(* CoDeSys 2.3 export: SCHU-P2-3.EXP *)

(* POU MAIN, CFC *)
PROGRAM MAIN
VAR
	TCT: ISTOK_TaskCycleTime;
END_VAR
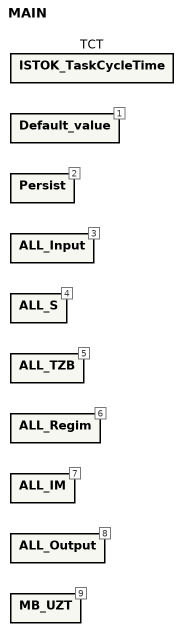
_CFC_ (* Continuous Function Chart, elements in execution order *)
#0 TCT:ISTOK_TaskCycleTime()
#1 Default_value()
#2 Persist()
#3 ALL_Input()
#4 ALL_S()
#5 ALL_TZB()
#6 ALL_Regim()
#7 ALL_IM()
#8 ALL_Output()
#9 MB_UZT()
_END_CFC_
(* the same logic as Structured Text *)
TCT();
Default_value();
Persist();
ALL_Input();
ALL_S();
ALL_TZB();
ALL_Regim();
ALL_IM();
ALL_Output();
MB_UZT();
END_PROGRAM

(* POU Lib/ISTOK_TaskCycleTime, CFC *)
FUNCTION_BLOCK ISTOK_TaskCycleTime
VAR_INPUT
END_VAR
VAR_OUTPUT
END_VAR
VAR
END_VAR
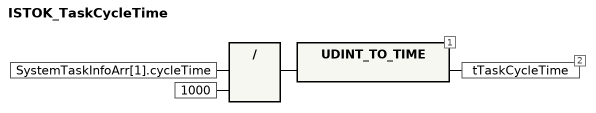
_CFC_ (* Continuous Function Chart, elements in execution order *)
#0 /(SystemTaskInfoArr[1].cycleTime, 1000)
#1 UDINT_TO_TIME(#0)
#2 tTaskCycleTime <= #1
_END_CFC_
END_FUNCTION_BLOCK

(* POU Default_value, CFC *)
PROGRAM Default_value
VAR
END_VAR
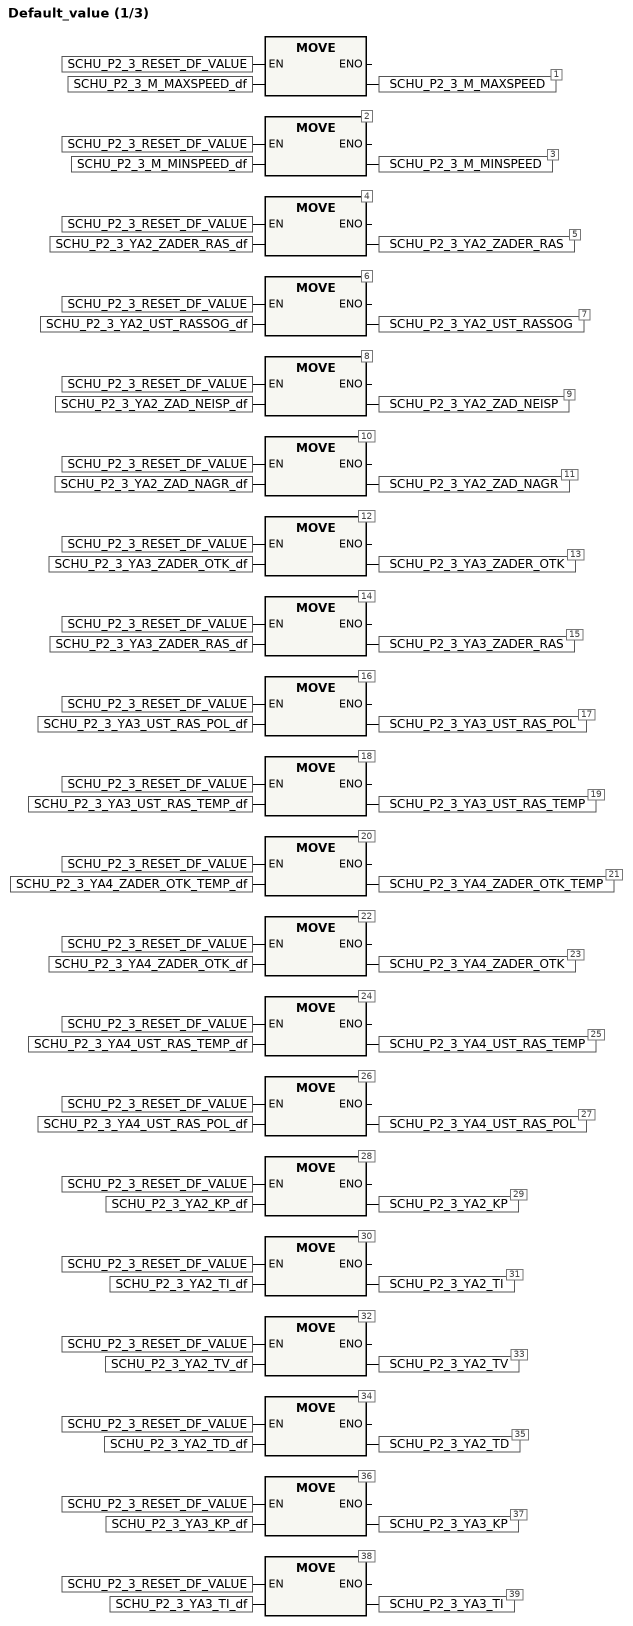
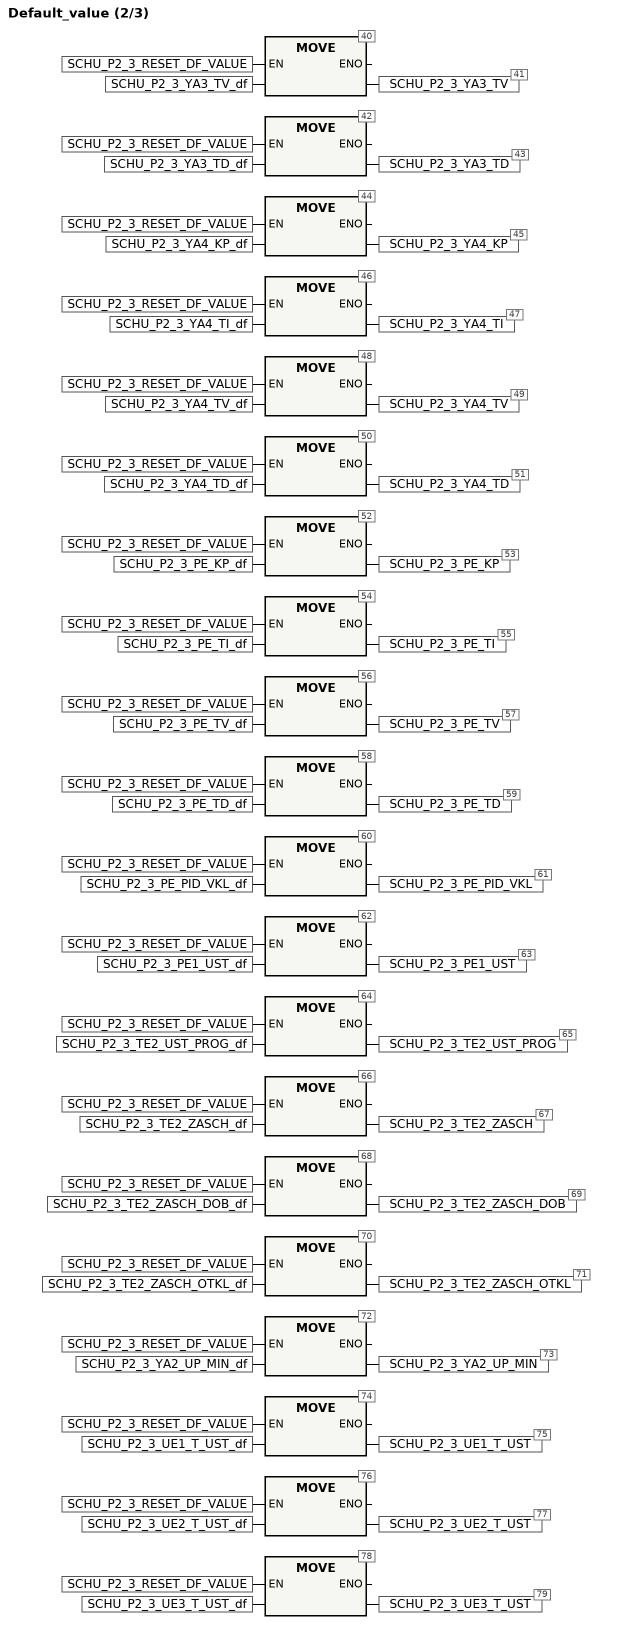
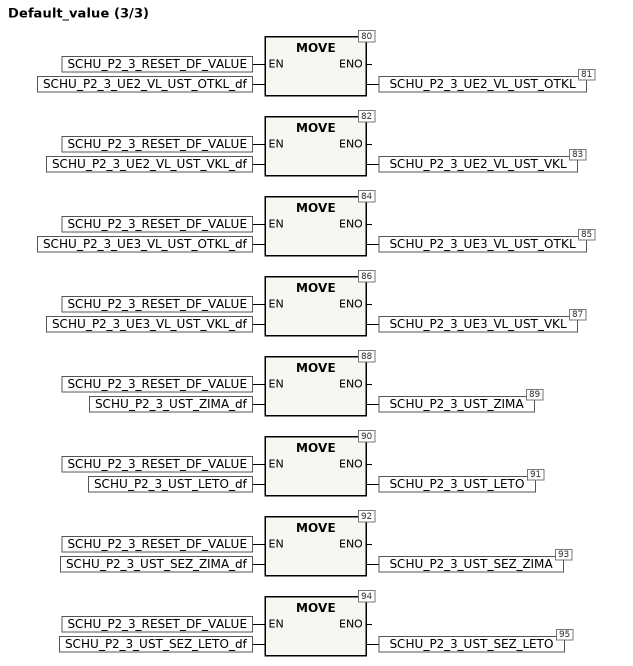
